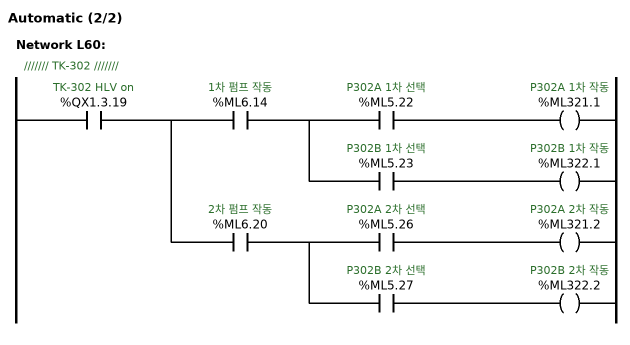
(* [picture p24: Automatic rungs L60-L60] *)
(* /////// TK-302 /////// *)
(* Rung L60 *)
%ML321.1 := %QX1.3.19 AND %ML6.14 AND %ML5.22;
%ML322.1 := %QX1.3.19 AND %ML6.14 AND %ML5.23;
%ML321.2 := %QX1.3.19 AND %ML6.20 AND %ML5.26;
%ML322.2 := %QX1.3.19 AND %ML6.20 AND %ML5.27;
END_PROGRAM

PROGRAM Analog (* task: 스캔 프로그램 *)
VAR_EXTERNAL
    _0100_CH0_ACT : BOOL; (* AT %UX1.0.16 *) (* 아날로그입력 모듈: 채널0 운전중 *)
    _0100_CH0_DATA : INT; (* AT %UW1.0.2 *) (* 아날로그입력 모듈: 채널0 변환값 *)
    _0100_CH0_IDD : BOOL; (* AT %UX1.0.160 *) (* 아날로그입력 모듈: 채널0 입력단선검출 *)
    _0100_CH1_ACT : BOOL; (* AT %UX1.0.17 *) (* 아날로그입력 모듈: 채널1 운전중 *)
    _0100_CH1_DATA : INT; (* AT %UW1.0.3 *) (* 아날로그입력 모듈: 채널1 변환값 *)
    _0100_CH1_IDD : BOOL; (* AT %UX1.0.161 *) (* 아날로그입력 모듈: 채널1 입력단선검출 *)
    _0100_CH2_ACT : BOOL; (* AT %UX1.0.18 *) (* 아날로그입력 모듈: 채널2 운전중 *)
    _0100_CH2_DATA : INT; (* AT %UW1.0.4 *) (* 아날로그입력 모듈: 채널2 변환값 *)
    _0100_CH2_IDD : BOOL; (* AT %UX1.0.162 *) (* 아날로그입력 모듈: 채널2 입력단선검출 *)
    _0100_CH3_ACT : BOOL; (* AT %UX1.0.19 *) (* 아날로그입력 모듈: 채널3 운전중 *)
    _0100_CH3_DATA : INT; (* AT %UW1.0.5 *) (* 아날로그입력 모듈: 채널3 변환값 *)
    _0100_CH3_IDD : BOOL; (* AT %UX1.0.163 *) (* 아날로그입력 모듈: 채널3 입력단선검출 *)
    _0100_CH4_ACT : BOOL; (* AT %UX1.0.20 *) (* 아날로그입력 모듈: 채널4 운전중 *)
    _0100_CH4_DATA : INT; (* AT %UW1.0.6 *) (* 아날로그입력 모듈: 채널4 변환값 *)
    _0100_CH4_IDD : BOOL; (* AT %UX1.0.164 *) (* 아날로그입력 모듈: 채널4 입력단선검출 *)
    _0100_CH5_ACT : BOOL; (* AT %UX1.0.21 *) (* 아날로그입력 모듈: 채널5 운전중 *)
    _0100_CH5_DATA : INT; (* AT %UW1.0.7 *) (* 아날로그입력 모듈: 채널5 변환값 *)
    _0100_CH5_IDD : BOOL; (* AT %UX1.0.165 *) (* 아날로그입력 모듈: 채널5 입력단선검출 *)
    _0100_CH6_ACT : BOOL; (* AT %UX1.0.22 *) (* 아날로그입력 모듈: 채널6 운전중 *)
    _0100_CH6_DATA : INT; (* AT %UW1.0.8 *) (* 아날로그입력 모듈: 채널6 변환값 *)
    _0100_CH6_IDD : BOOL; (* AT %UX1.0.166 *) (* 아날로그입력 모듈: 채널6 입력단선검출 *)
END_VAR
VAR
    _t1 : BOOL;
    _t2 : BOOL;
    _t3 : BOOL;
    _t4 : BOOL;
    _t5 : BOOL;
    _t6 : BOOL;
    _t7 : BOOL;
    _t8 : BOOL;
    _t9 : BOOL;
END_VAR

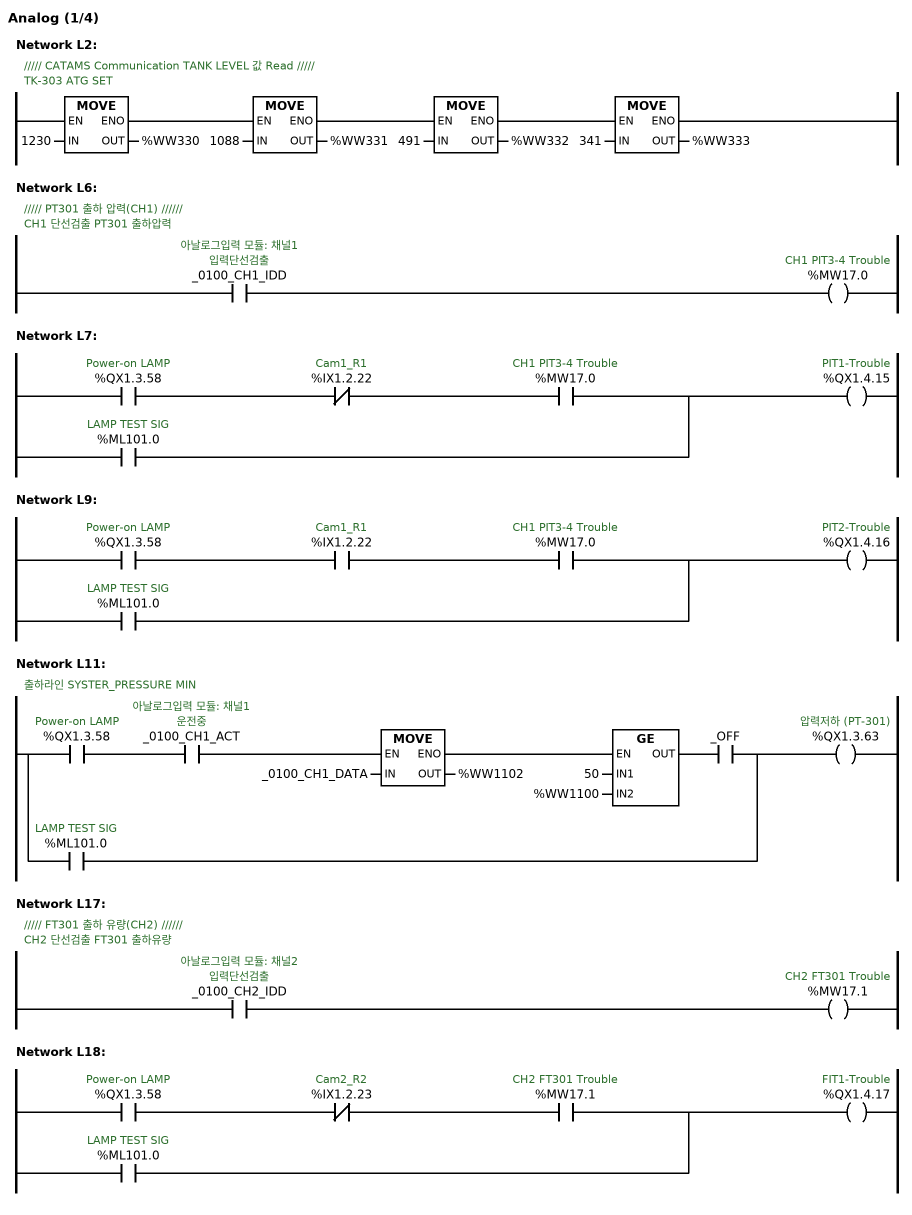
(* ///// CATAMS Communication TANK LEVEL 값 Read ///// *)
(* TK-303 ATG SET *)
(* Rung L2 *)
%WW330 := 1230;
%WW331 := 1088;
%WW332 := 491;
%WW333 := 341;
(* ///// PT301 출하 압력(CH1) ////// *)
(* Rung L6 *)
%MW17.0 := _0100_CH1_IDD;
(* CH1 단선검출 PT301 출하압력 *)
(* Rung L7 *)
%QX1.4.15 := (%QX1.3.58 AND NOT %IX1.2.22 AND %MW17.0) OR %ML101.0;
(* Rung L9 *)
%QX1.4.16 := (%QX1.3.58 AND %IX1.2.22 AND %MW17.0) OR %ML101.0;
(* Rung L11 *)
IF %QX1.3.58 AND _0100_CH1_ACT THEN
    %WW1102 := _0100_CH1_DATA;
    _t1 := 50 >= %WW1100;
END_IF;
%QX1.3.63 := (_t1 AND _OFF) OR %ML101.0;
(* 출하라인 SYSTER_PRESSURE MIN *)
(* ///// FT301 출하 유량(CH2) ////// *)
(* Rung L17 *)
%MW17.1 := _0100_CH2_IDD;
(* CH2 단선검출 FT301 출하유량 *)
(* Rung L18 *)
%QX1.4.17 := (%QX1.3.58 AND NOT %IX1.2.23 AND %MW17.1) OR %ML101.0;

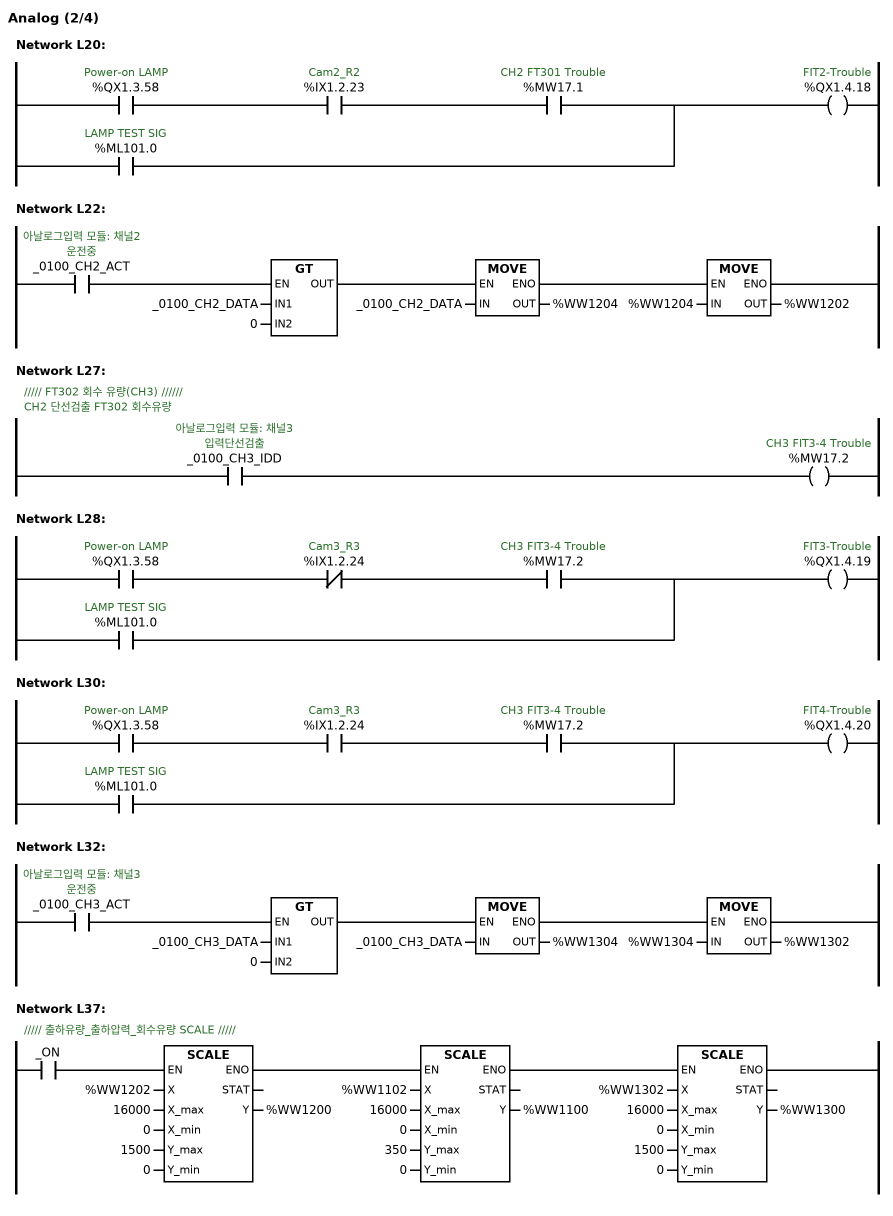
(* Rung L20 *)
%QX1.4.18 := (%QX1.3.58 AND %IX1.2.23 AND %MW17.1) OR %ML101.0;
(* Rung L22 *)
IF _0100_CH2_ACT THEN _t2 := _0100_CH2_DATA > 0; END_IF;
IF _t2 THEN
    %WW1204 := _0100_CH2_DATA;
    %WW1202 := %WW1204;
END_IF;
(* ///// FT302 회수 유량(CH3) ////// *)
(* Rung L27 *)
%MW17.2 := _0100_CH3_IDD;
(* CH2 단선검출 FT302 회수유량 *)
(* Rung L28 *)
%QX1.4.19 := (%QX1.3.58 AND NOT %IX1.2.24 AND %MW17.2) OR %ML101.0;
(* Rung L30 *)
%QX1.4.20 := (%QX1.3.58 AND %IX1.2.24 AND %MW17.2) OR %ML101.0;
(* Rung L32 *)
IF _0100_CH3_ACT THEN _t3 := _0100_CH3_DATA > 0; END_IF;
IF _t3 THEN
    %WW1304 := _0100_CH3_DATA;
    %WW1302 := %WW1304;
END_IF;
(* ///// 출하유량_출하압력_회수유량 SCALE ///// *)
(* Rung L37 *)
IF _ON THEN
    SCALE(X := %WW1202, X_max := 16000, X_min := 0, Y_max := 1500, Y_min := 0, Y => %WW1200);
    SCALE(X := %WW1102, X_max := 16000, X_min := 0, Y_max := 350, Y_min := 0, Y => %WW1100);
    SCALE(X := %WW1302, X_max := 16000, X_min := 0, Y_max := 1500, Y_min := 0, Y => %WW1300);
END_IF;

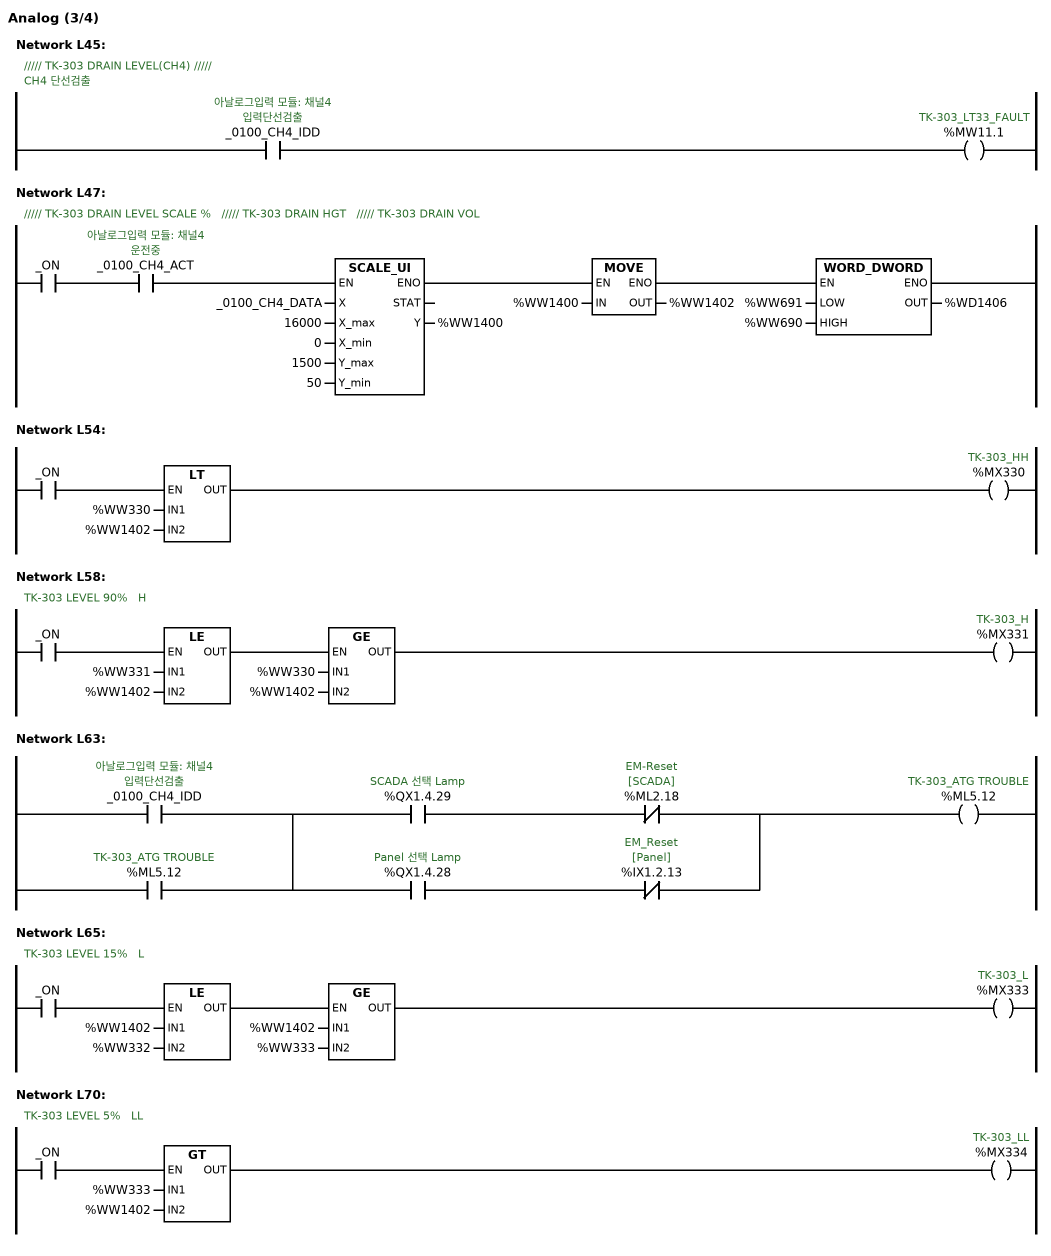
(* ///// TK-303 DRAIN LEVEL(CH4) ///// *)
(* Rung L45 *)
%MW11.1 := _0100_CH4_IDD;
(* CH4 단선검출 *)
(* ///// TK-303 DRAIN LEVEL SCALE %   ///// TK-303 DRAIN HGT   ///// TK-303 DRAIN VOL *)
(* Rung L47 *)
IF _ON AND _0100_CH4_ACT THEN
    SCALE_UI(X := _0100_CH4_DATA, X_max := 16000, X_min := 0, Y_max := 1500, Y_min := 50, Y => %WW1400);
    %WW1402 := %WW1400;
    %WD1406 := WORD_DWORD(LOW := %WW691, HIGH := %WW690);
END_IF;
(* Rung L54 *)
IF _ON THEN _t4 := %WW330 < %WW1402; END_IF;
%MX330 := _t4;
(* Rung L58 *)
IF _ON THEN _t5 := %WW331 <= %WW1402; END_IF;
IF _t5 THEN _t6 := %WW330 >= %WW1402; END_IF;
%MX331 := _t6;
(* TK-303 LEVEL 90%   H *)
(* Rung L63 *)
%ML5.12 := (_0100_CH4_IDD OR %ML5.12) AND ((%QX1.4.29 AND NOT %ML2.18) OR (%QX1.4.28 AND NOT %IX1.2.13));
(* Rung L65 *)
IF _ON THEN _t7 := %WW1402 <= %WW332; END_IF;
IF _t7 THEN _t8 := %WW1402 >= %WW333; END_IF;
%MX333 := _t8;
(* TK-303 LEVEL 15%   L *)
(* Rung L70 *)
IF _ON THEN _t9 := %WW333 > %WW1402; END_IF;
%MX334 := _t9;
(* TK-303 LEVEL 5%   LL *)

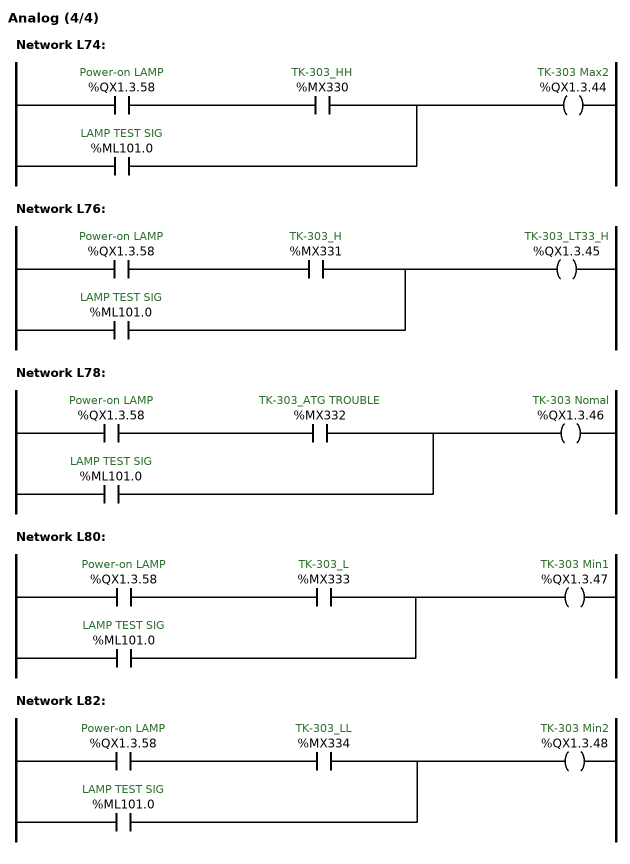
(* Rung L74 *)
%QX1.3.44 := (%QX1.3.58 AND %MX330) OR %ML101.0;
(* Rung L76 *)
%QX1.3.45 := (%QX1.3.58 AND %MX331) OR %ML101.0;
(* Rung L78 *)
%QX1.3.46 := (%QX1.3.58 AND %MX332) OR %ML101.0;
(* Rung L80 *)
%QX1.3.47 := (%QX1.3.58 AND %MX333) OR %ML101.0;
(* Rung L82 *)
%QX1.3.48 := (%QX1.3.58 AND %MX334) OR %ML101.0;
END_PROGRAM

PROGRAM Communiction (* task: 스캔 프로그램 *)
VAR
    C0010 : CTR; (* 통신 *)
    C19_TLV_OFD : TOF;
    C20_TLV_OFD : TOF;
    C21_TLV_OFD : TOF;
    C22_TLV_OFD : TOF;
    C23_TLV_OFD : TOF;
    C24_TLV_OFD : TOF;
    C24_TLV_OFD1 : TON;
    C24_TLV_OFD2 : TON;
    C24_TLV_OFD3 : TOF;
    C24_TLV_OFD4 : TOF;
    C24_TLV_OFD5 : TON;
    CTR10 : BOOL; (* 모드버스 송신블럭 번호 *)
END_VAR
VAR_EXTERNAL
    _0100_CH1_ACT : BOOL; (* AT %UX1.0.17 *) (* 아날로그입력 모듈: 채널1 운전중 *)
    _0100_CH1_DATA : INT; (* AT %UW1.0.3 *) (* 아날로그입력 모듈: 채널1 변환값 *)
END_VAR
VAR
    _t1 : BOOL;
    _t2 : BOOL;
    _t3 : BOOL;
    _t4 : BOOL;
    _t5 : BOOL;
    _t6 : BOOL;
    _t7 : BOOL;
    _t8 : BOOL;
    _t9 : BOOL;
    _t10 : BOOL;
    _t11 : BOOL;
    _t12 : BOOL;
    _t13 : BOOL;
    _t14 : BOOL;
END_VAR

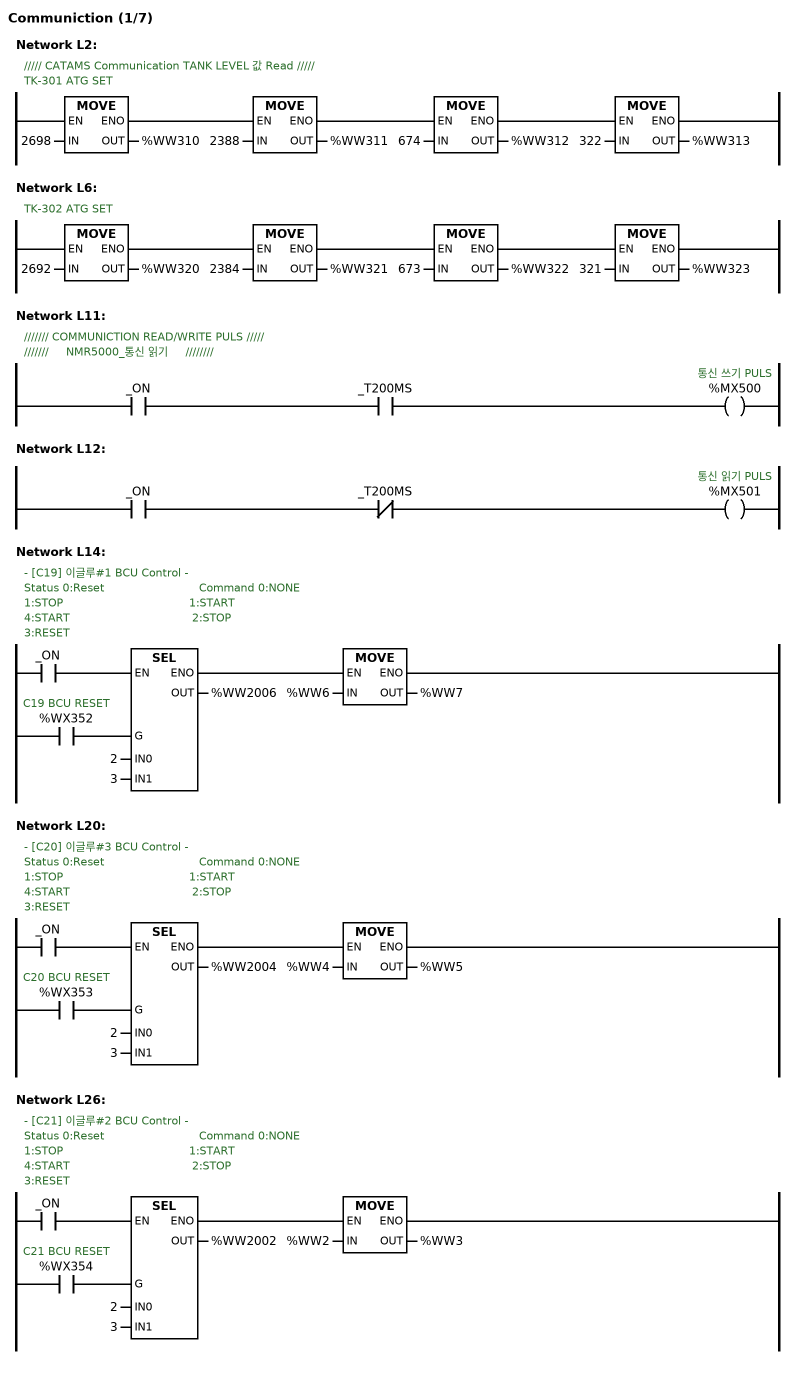
(* ///// CATAMS Communication TANK LEVEL 값 Read ///// *)
(* TK-301 ATG SET *)
(* Rung L2 *)
%WW310 := 2698;
%WW311 := 2388;
%WW312 := 674;
%WW313 := 322;
(* TK-302 ATG SET *)
(* Rung L6 *)
%WW320 := 2692;
%WW321 := 2384;
%WW322 := 673;
%WW323 := 321;
(* /////// COMMUNICTION READ/WRITE PULS ///// *)
(* ///////     NMR5000_통신 읽기     //////// *)
(* Rung L11 *)
%MX500 := _ON AND _T200MS;
(* Rung L12 *)
%MX501 := _ON AND NOT _T200MS;
(* - [C19] 이글루#1 BCU Control - / Status 0:Reset                           Command 0:NONE / 1:STOP                                    1:START / 4:START                                   2:STOP / 3:RESET *)
(* Rung L14 *)
IF _ON THEN
    %WW2006 := SEL(G := %WX352, IN0 := 2, IN1 := 3);
    %WW7 := %WW6;
END_IF;
(* - [C20] 이글루#3 BCU Control - / Status 0:Reset                           Command 0:NONE / 1:STOP                                    1:START / 4:START                                   2:STOP / 3:RESET *)
(* Rung L20 *)
IF _ON THEN
    %WW2004 := SEL(G := %WX353, IN0 := 2, IN1 := 3);
    %WW5 := %WW4;
END_IF;
(* - [C21] 이글루#2 BCU Control - / Status 0:Reset                           Command 0:NONE / 1:STOP                                    1:START / 4:START                                   2:STOP / 3:RESET *)
(* Rung L26 *)
IF _ON THEN
    %WW2002 := SEL(G := %WX354, IN0 := 2, IN1 := 3);
    %WW3 := %WW2;
END_IF;

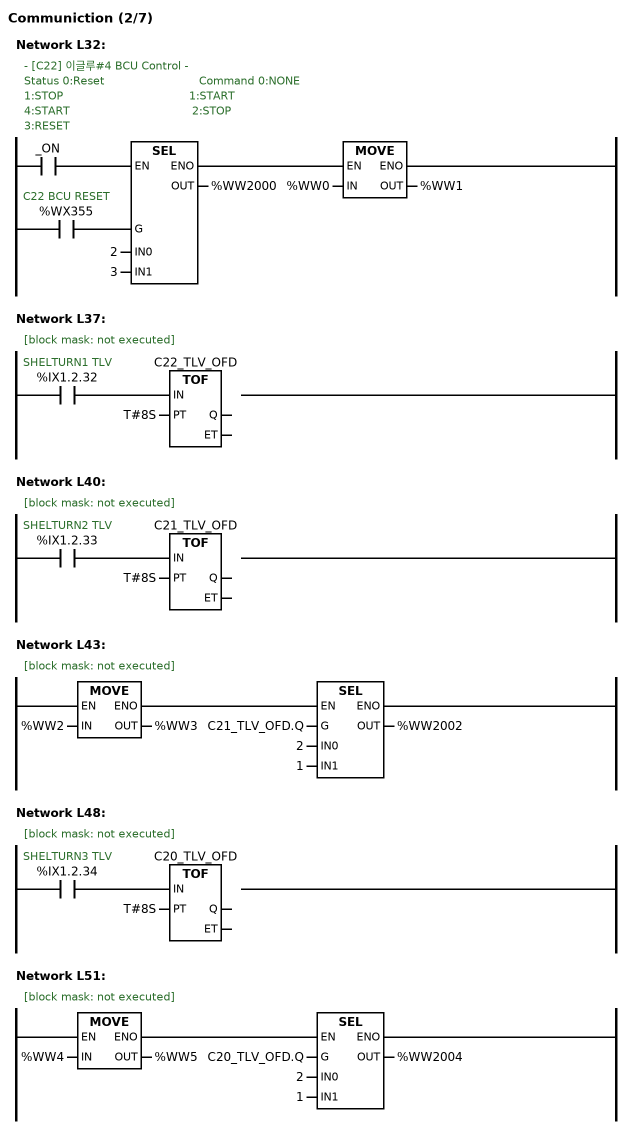
(* - [C22] 이글루#4 BCU Control - / Status 0:Reset                           Command 0:NONE / 1:STOP                                    1:START / 4:START                                   2:STOP / 3:RESET *)
(* Rung L32 *)
IF _ON THEN
    %WW2000 := SEL(G := %WX355, IN0 := 2, IN1 := 3);
    %WW1 := %WW0;
END_IF;
(* Rung L37 is block-masked: not executed *)
// C22_TLV_OFD(IN := %IX1.2.32, PT := T#8S);
(* Rung L40 is block-masked: not executed *)
// C21_TLV_OFD(IN := %IX1.2.33, PT := T#8S);
(* Rung L43 is block-masked: not executed *)
// %WW3 := %WW2;
// %WW2002 := SEL(G := C21_TLV_OFD.Q, IN0 := 2, IN1 := 1);
(* Rung L48 is block-masked: not executed *)
// C20_TLV_OFD(IN := %IX1.2.34, PT := T#8S);
(* Rung L51 is block-masked: not executed *)
// %WW5 := %WW4;
// %WW2004 := SEL(G := C20_TLV_OFD.Q, IN0 := 2, IN1 := 1);

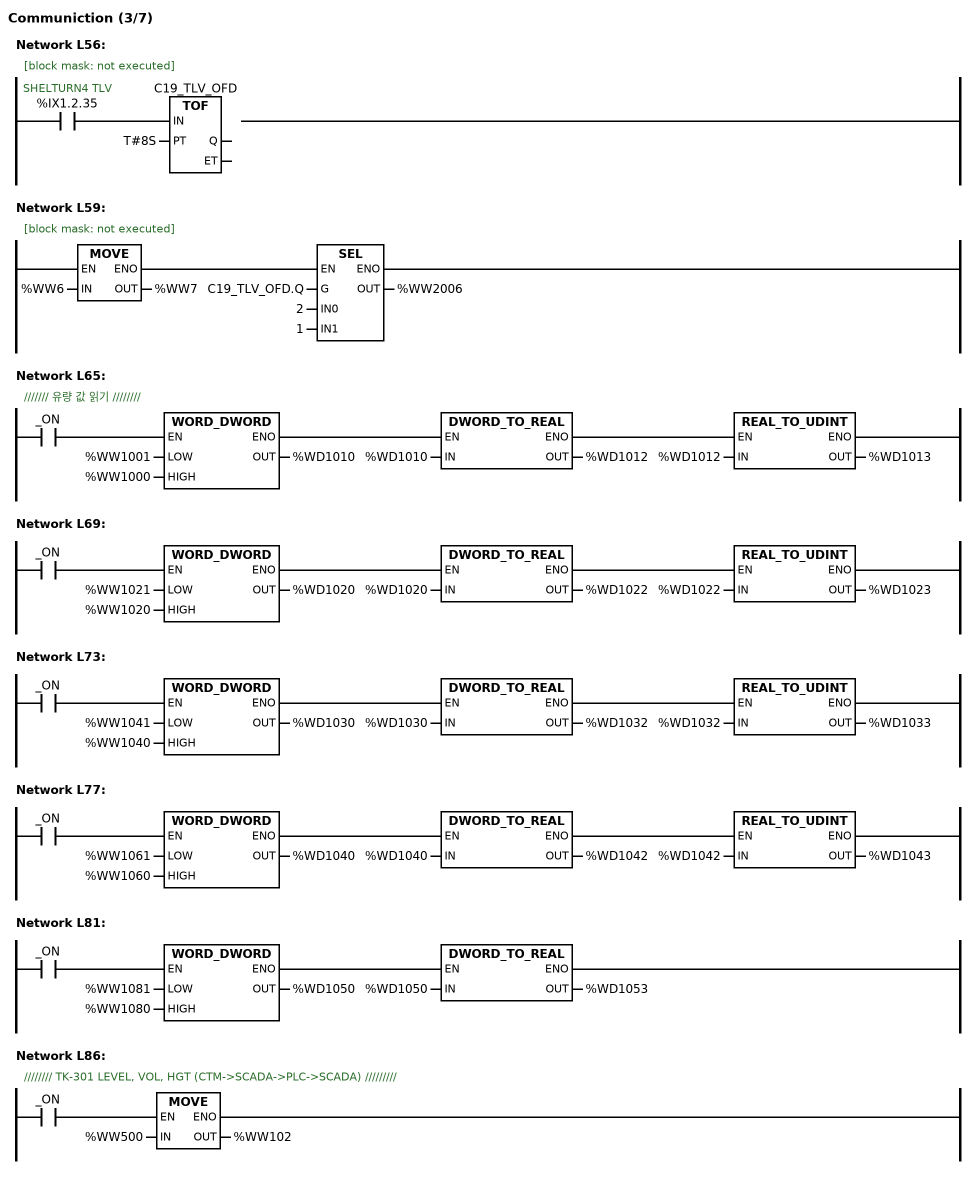
(* Rung L56 is block-masked: not executed *)
// C19_TLV_OFD(IN := %IX1.2.35, PT := T#8S);
(* Rung L59 is block-masked: not executed *)
// %WW7 := %WW6;
// %WW2006 := SEL(G := C19_TLV_OFD.Q, IN0 := 2, IN1 := 1);
(* /////// 유량 값 읽기 //////// *)
(* Rung L65 *)
IF _ON THEN
    %WD1010 := WORD_DWORD(LOW := %WW1001, HIGH := %WW1000);
    %WD1012 := DWORD_TO_REAL(%WD1010);
    %WD1013 := REAL_TO_UDINT(%WD1012);
END_IF;
(* Rung L69 *)
IF _ON THEN
    %WD1020 := WORD_DWORD(LOW := %WW1021, HIGH := %WW1020);
    %WD1022 := DWORD_TO_REAL(%WD1020);
    %WD1023 := REAL_TO_UDINT(%WD1022);
END_IF;
(* Rung L73 *)
IF _ON THEN
    %WD1030 := WORD_DWORD(LOW := %WW1041, HIGH := %WW1040);
    %WD1032 := DWORD_TO_REAL(%WD1030);
    %WD1033 := REAL_TO_UDINT(%WD1032);
END_IF;
(* Rung L77 *)
IF _ON THEN
    %WD1040 := WORD_DWORD(LOW := %WW1061, HIGH := %WW1060);
    %WD1042 := DWORD_TO_REAL(%WD1040);
    %WD1043 := REAL_TO_UDINT(%WD1042);
END_IF;
(* Rung L81 *)
IF _ON THEN
    %WD1050 := WORD_DWORD(LOW := %WW1081, HIGH := %WW1080);
    %WD1053 := DWORD_TO_REAL(%WD1050);
END_IF;
(* //////// TK-301 LEVEL, VOL, HGT (CTM->SCADA->PLC->SCADA) ///////// *)
(* Rung L86 *)
IF _ON THEN %WW102 := %WW500; END_IF;

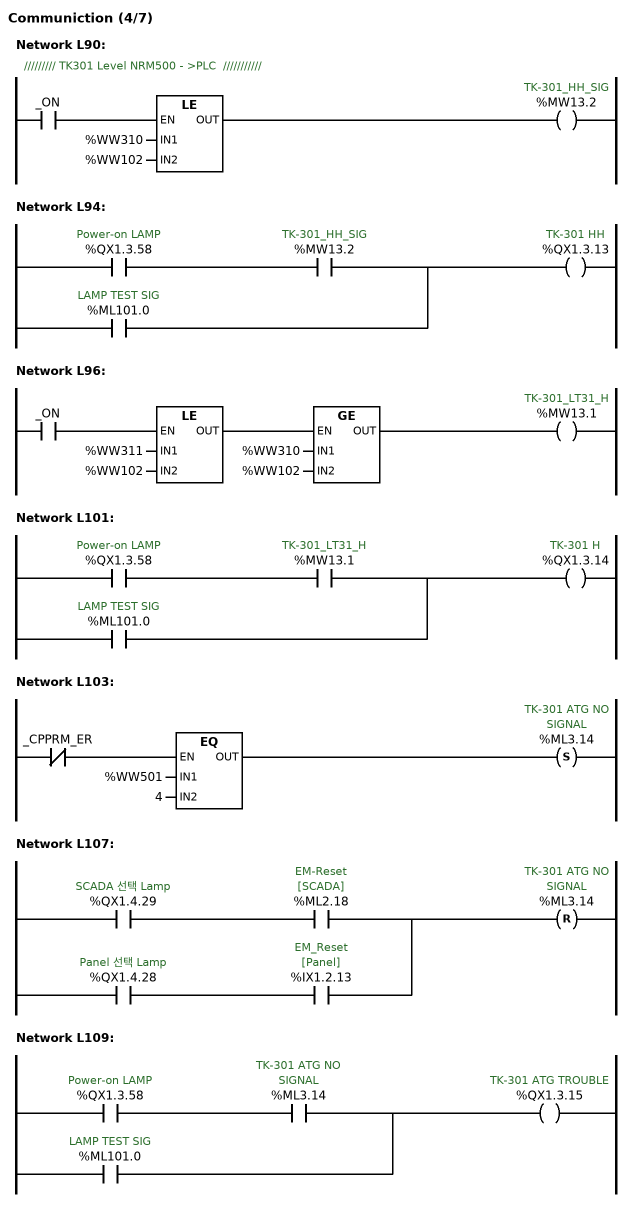
(* ///////// TK301 Level NRM500 - >PLC  /////////// *)
(* Rung L90 *)
IF _ON THEN _t1 := %WW310 <= %WW102; END_IF;
%MW13.2 := _t1;
(* Rung L94 *)
%QX1.3.13 := (%QX1.3.58 AND %MW13.2) OR %ML101.0;
(* Rung L96 *)
IF _ON THEN _t2 := %WW311 <= %WW102; END_IF;
IF _t2 THEN _t3 := %WW310 >= %WW102; END_IF;
%MW13.1 := _t3;
(* Rung L101 *)
%QX1.3.14 := (%QX1.3.58 AND %MW13.1) OR %ML101.0;
(* Rung L103 *)
IF NOT _CPPRM_ER THEN _t4 := %WW501 = 4; END_IF;
IF _t4 THEN %ML3.14 := TRUE; END_IF;
(* Rung L107 *)
IF (%QX1.4.29 AND %ML2.18) OR (%QX1.4.28 AND %IX1.2.13) THEN %ML3.14 := FALSE; END_IF;
(* Rung L109 *)
%QX1.3.15 := (%QX1.3.58 AND %ML3.14) OR %ML101.0;

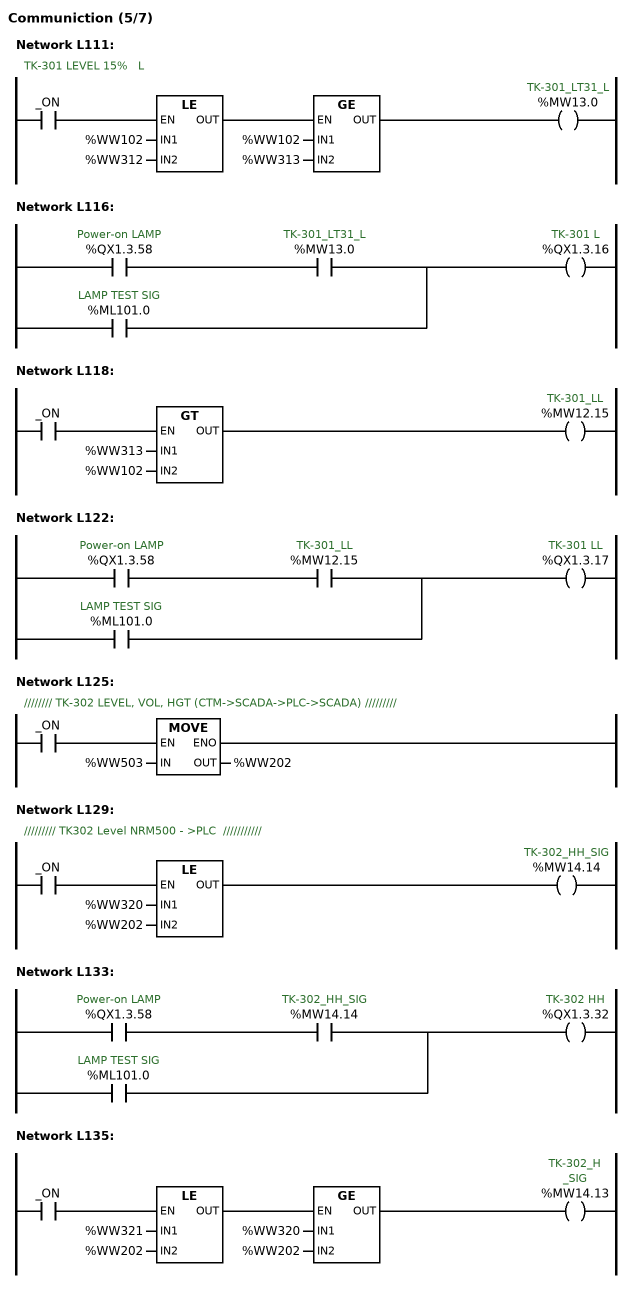
(* Rung L111 *)
IF _ON THEN _t5 := %WW102 <= %WW312; END_IF;
IF _t5 THEN _t6 := %WW102 >= %WW313; END_IF;
%MW13.0 := _t6;
(* TK-301 LEVEL 15%   L *)
(* Rung L116 *)
%QX1.3.16 := (%QX1.3.58 AND %MW13.0) OR %ML101.0;
(* Rung L118 *)
IF _ON THEN _t7 := %WW313 > %WW102; END_IF;
%MW12.15 := _t7;
(* Rung L122 *)
%QX1.3.17 := (%QX1.3.58 AND %MW12.15) OR %ML101.0;
(* //////// TK-302 LEVEL, VOL, HGT (CTM->SCADA->PLC->SCADA) ///////// *)
(* Rung L125 *)
IF _ON THEN %WW202 := %WW503; END_IF;
(* ///////// TK302 Level NRM500 - >PLC  /////////// *)
(* Rung L129 *)
IF _ON THEN _t8 := %WW320 <= %WW202; END_IF;
%MW14.14 := _t8;
(* Rung L133 *)
%QX1.3.32 := (%QX1.3.58 AND %MW14.14) OR %ML101.0;
(* Rung L135 *)
IF _ON THEN _t9 := %WW321 <= %WW202; END_IF;
IF _t9 THEN _t10 := %WW320 >= %WW202; END_IF;
%MW14.13 := _t10;

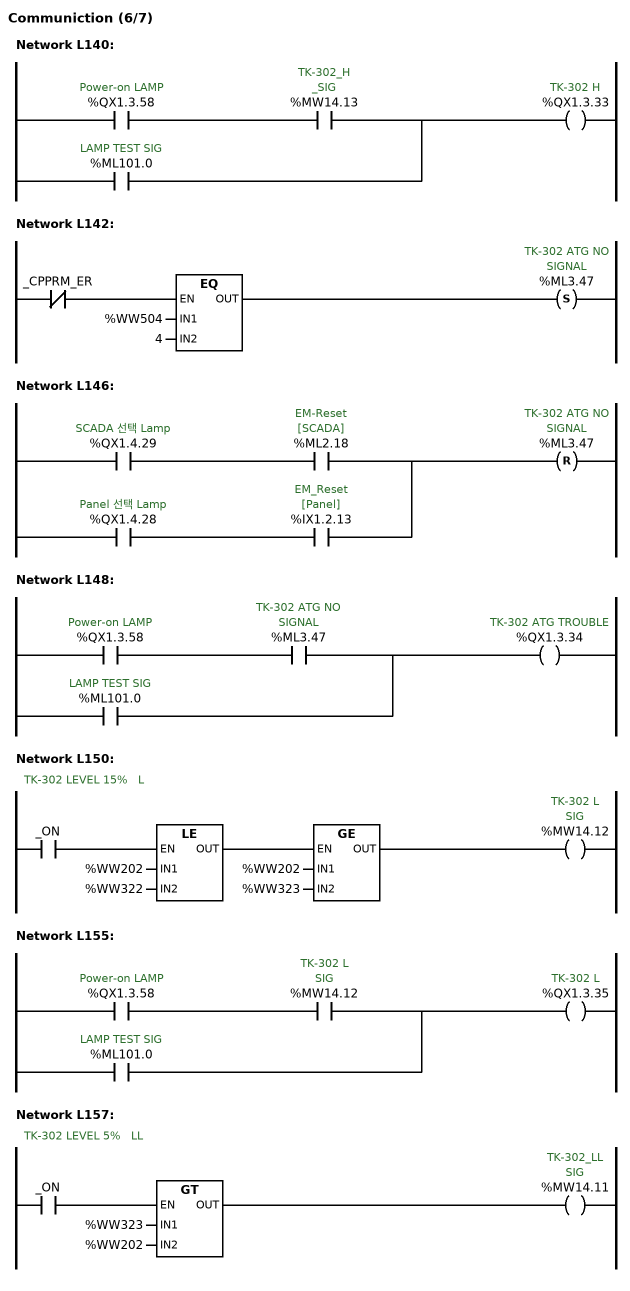
(* Rung L140 *)
%QX1.3.33 := (%QX1.3.58 AND %MW14.13) OR %ML101.0;
(* Rung L142 *)
IF NOT _CPPRM_ER THEN _t11 := %WW504 = 4; END_IF;
IF _t11 THEN %ML3.47 := TRUE; END_IF;
(* Rung L146 *)
IF (%QX1.4.29 AND %ML2.18) OR (%QX1.4.28 AND %IX1.2.13) THEN %ML3.47 := FALSE; END_IF;
(* Rung L148 *)
%QX1.3.34 := (%QX1.3.58 AND %ML3.47) OR %ML101.0;
(* Rung L150 *)
IF _ON THEN _t12 := %WW202 <= %WW322; END_IF;
IF _t12 THEN _t13 := %WW202 >= %WW323; END_IF;
%MW14.12 := _t13;
(* TK-302 LEVEL 15%   L *)
(* Rung L155 *)
%QX1.3.35 := (%QX1.3.58 AND %MW14.12) OR %ML101.0;
(* Rung L157 *)
IF _ON THEN _t14 := %WW323 > %WW202; END_IF;
%MW14.11 := _t14;
(* TK-302 LEVEL 5%   LL *)

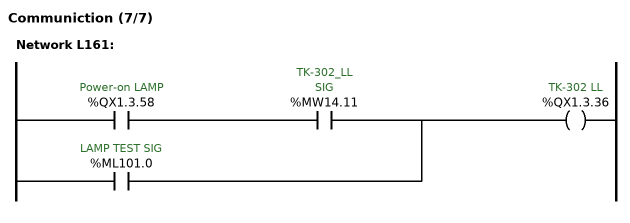
(* Rung L161 *)
%QX1.3.36 := (%QX1.3.58 AND %MW14.11) OR %ML101.0;
END_PROGRAM

PROGRAM Scada (* task: 스캔 프로그램 *)
VAR
    T1 : BOOL;
    T9 : TON;
END_VAR

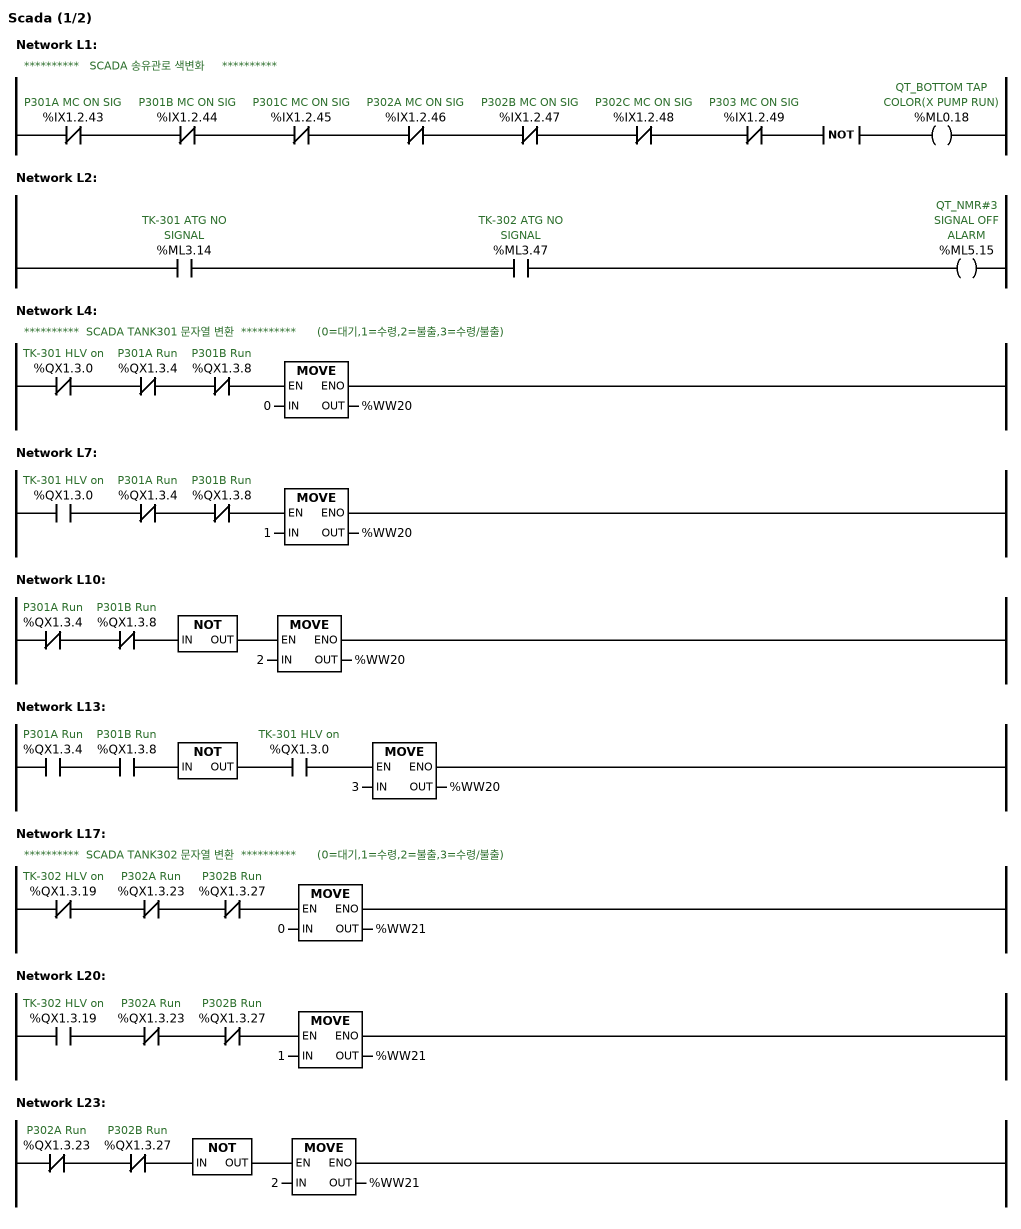
(* **********   SCADA 송유관로 색변화     ********** *)
(* Rung L1 *)
%ML0.18 := NOT (NOT %IX1.2.43 AND NOT %IX1.2.44 AND NOT %IX1.2.45 AND NOT %IX1.2.46 AND NOT %IX1.2.47 AND NOT %IX1.2.48 AND NOT %IX1.2.49);
(* Rung L2 *)
%ML5.15 := %ML3.14 AND %ML3.47;
(* **********  SCADA TANK301 문자열 변환  **********      (0=대기,1=수령,2=불출,3=수령/불출) *)
(* Rung L4 *)
IF NOT %QX1.3.0 AND NOT %QX1.3.4 AND NOT %QX1.3.8 THEN %WW20 := 0; END_IF;
(* Rung L7 *)
IF %QX1.3.0 AND NOT %QX1.3.4 AND NOT %QX1.3.8 THEN %WW20 := 1; END_IF;
(* Rung L10 *)
IF NOT (NOT %QX1.3.4 AND NOT %QX1.3.8) THEN %WW20 := 2; END_IF;
(* Rung L13 *)
IF (NOT (%QX1.3.4 AND %QX1.3.8)) AND %QX1.3.0 THEN %WW20 := 3; END_IF;
(* **********  SCADA TANK302 문자열 변환  **********      (0=대기,1=수령,2=불출,3=수령/불출) *)
(* Rung L17 *)
IF NOT %QX1.3.19 AND NOT %QX1.3.23 AND NOT %QX1.3.27 THEN %WW21 := 0; END_IF;
(* Rung L20 *)
IF %QX1.3.19 AND NOT %QX1.3.23 AND NOT %QX1.3.27 THEN %WW21 := 1; END_IF;
(* Rung L23 *)
IF NOT (NOT %QX1.3.23 AND NOT %QX1.3.27) THEN %WW21 := 2; END_IF;

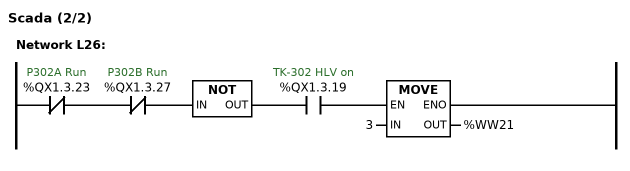
(* Rung L26 *)
IF (NOT (NOT %QX1.3.23 AND NOT %QX1.3.27)) AND %QX1.3.19 THEN %WW21 := 3; END_IF;
END_PROGRAM

PROGRAM Setting (* task: 스캔 프로그램 *)
VAR
    _t1 : BOOL;
    _t2 : BOOL;
    _t3 : BOOL;
    _t4 : BOOL;
    _t5 : BOOL;
    _t6 : BOOL;
    _t7 : BOOL;
    _t8 : BOOL;
END_VAR

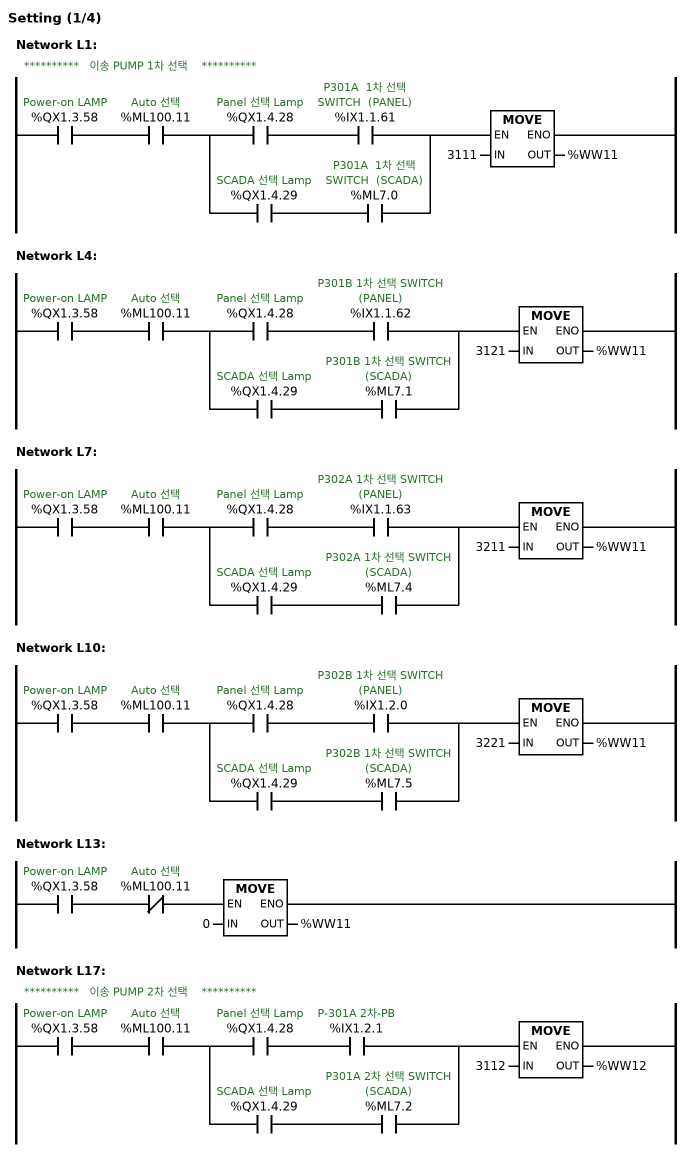
(* **********   이송 PUMP 1차 선택    ********** *)
(* Rung L1 *)
IF %QX1.3.58 AND %ML100.11 AND ((%QX1.4.28 AND %IX1.1.61) OR (%QX1.4.29 AND %ML7.0)) THEN
    %WW11 := 3111;
END_IF;
(* Rung L4 *)
IF %QX1.3.58 AND %ML100.11 AND ((%QX1.4.28 AND %IX1.1.62) OR (%QX1.4.29 AND %ML7.1)) THEN
    %WW11 := 3121;
END_IF;
(* Rung L7 *)
IF %QX1.3.58 AND %ML100.11 AND ((%QX1.4.28 AND %IX1.1.63) OR (%QX1.4.29 AND %ML7.4)) THEN
    %WW11 := 3211;
END_IF;
(* Rung L10 *)
IF %QX1.3.58 AND %ML100.11 AND ((%QX1.4.28 AND %IX1.2.0) OR (%QX1.4.29 AND %ML7.5)) THEN
    %WW11 := 3221;
END_IF;
(* Rung L13 *)
IF %QX1.3.58 AND NOT %ML100.11 THEN %WW11 := 0; END_IF;
(* **********   이송 PUMP 2차 선택    ********** *)
(* Rung L17 *)
IF %QX1.3.58 AND %ML100.11 AND ((%QX1.4.28 AND %IX1.2.1) OR (%QX1.4.29 AND %ML7.2)) THEN
    %WW12 := 3112;
END_IF;

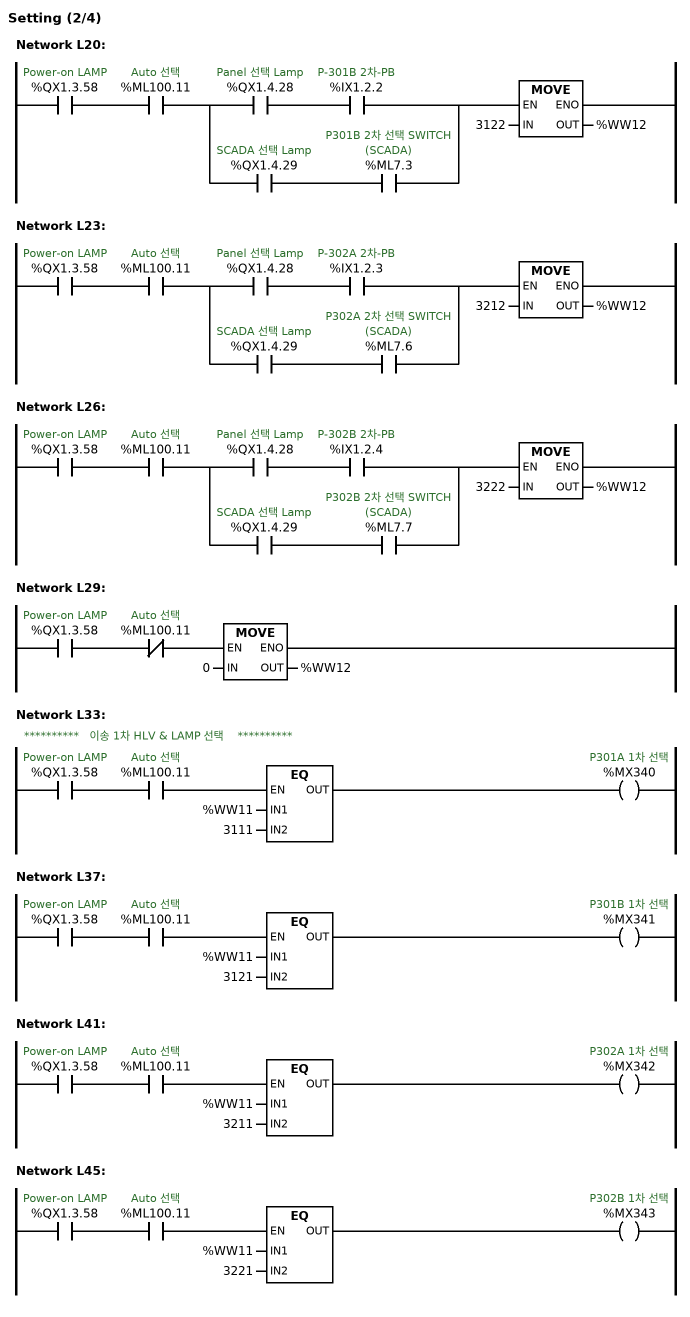
(* Rung L20 *)
IF %QX1.3.58 AND %ML100.11 AND ((%QX1.4.28 AND %IX1.2.2) OR (%QX1.4.29 AND %ML7.3)) THEN
    %WW12 := 3122;
END_IF;
(* Rung L23 *)
IF %QX1.3.58 AND %ML100.11 AND ((%QX1.4.28 AND %IX1.2.3) OR (%QX1.4.29 AND %ML7.6)) THEN
    %WW12 := 3212;
END_IF;
(* Rung L26 *)
IF %QX1.3.58 AND %ML100.11 AND ((%QX1.4.28 AND %IX1.2.4) OR (%QX1.4.29 AND %ML7.7)) THEN
    %WW12 := 3222;
END_IF;
(* Rung L29 *)
IF %QX1.3.58 AND NOT %ML100.11 THEN %WW12 := 0; END_IF;
(* **********   이송 1차 HLV & LAMP 선택    ********** *)
(* Rung L33 *)
IF %QX1.3.58 AND %ML100.11 THEN _t1 := %WW11 = 3111; END_IF;
%MX340 := _t1;
(* Rung L37 *)
IF %QX1.3.58 AND %ML100.11 THEN _t2 := %WW11 = 3121; END_IF;
%MX341 := _t2;
(* Rung L41 *)
IF %QX1.3.58 AND %ML100.11 THEN _t3 := %WW11 = 3211; END_IF;
%MX342 := _t3;
(* Rung L45 *)
IF %QX1.3.58 AND %ML100.11 THEN _t4 := %WW11 = 3221; END_IF;
%MX343 := _t4;

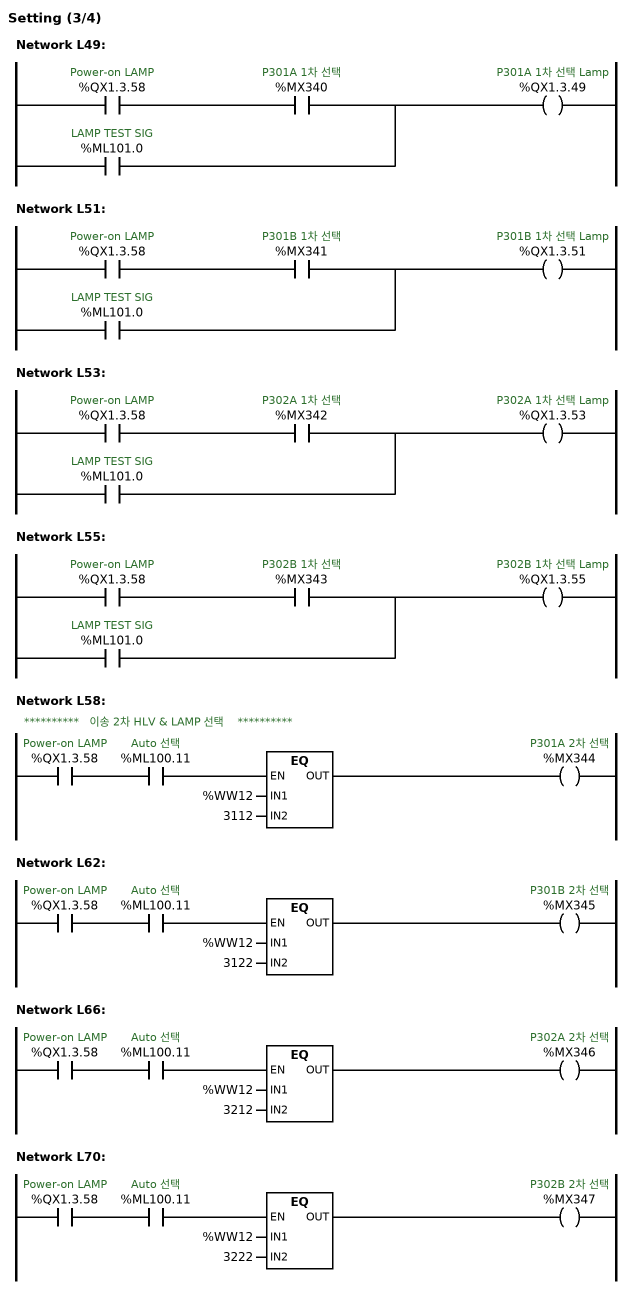
(* Rung L49 *)
%QX1.3.49 := (%QX1.3.58 AND %MX340) OR %ML101.0;
(* Rung L51 *)
%QX1.3.51 := (%QX1.3.58 AND %MX341) OR %ML101.0;
(* Rung L53 *)
%QX1.3.53 := (%QX1.3.58 AND %MX342) OR %ML101.0;
(* Rung L55 *)
%QX1.3.55 := (%QX1.3.58 AND %MX343) OR %ML101.0;
(* **********   이송 2차 HLV & LAMP 선택    ********** *)
(* Rung L58 *)
IF %QX1.3.58 AND %ML100.11 THEN _t5 := %WW12 = 3112; END_IF;
%MX344 := _t5;
(* Rung L62 *)
IF %QX1.3.58 AND %ML100.11 THEN _t6 := %WW12 = 3122; END_IF;
%MX345 := _t6;
(* Rung L66 *)
IF %QX1.3.58 AND %ML100.11 THEN _t7 := %WW12 = 3212; END_IF;
%MX346 := _t7;
(* Rung L70 *)
IF %QX1.3.58 AND %ML100.11 THEN _t8 := %WW12 = 3222; END_IF;
%MX347 := _t8;

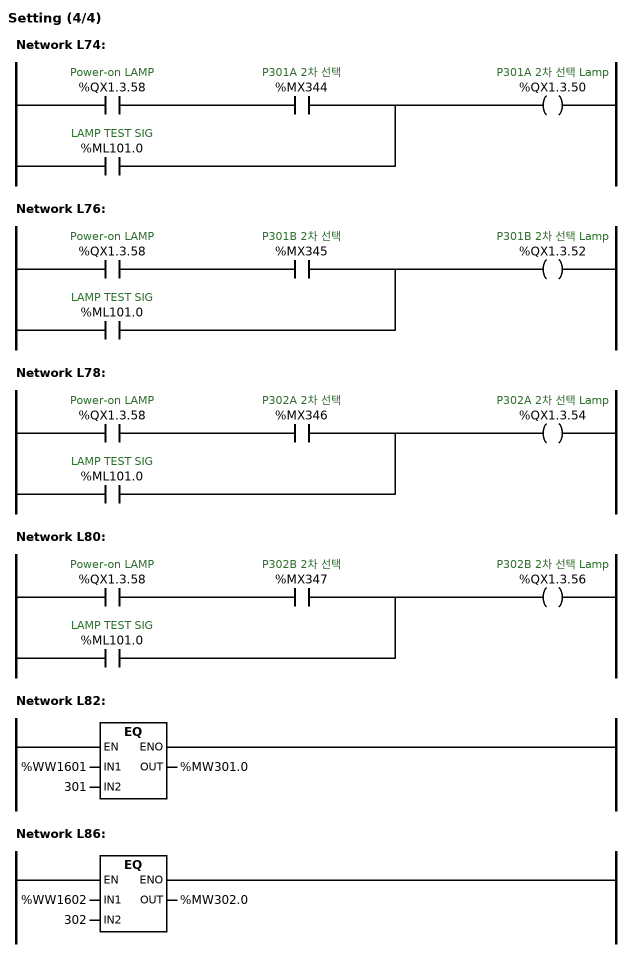
(* Rung L74 *)
%QX1.3.50 := (%QX1.3.58 AND %MX344) OR %ML101.0;
(* Rung L76 *)
%QX1.3.52 := (%QX1.3.58 AND %MX345) OR %ML101.0;
(* Rung L78 *)
%QX1.3.54 := (%QX1.3.58 AND %MX346) OR %ML101.0;
(* Rung L80 *)
%QX1.3.56 := (%QX1.3.58 AND %MX347) OR %ML101.0;
(* Rung L82 *)
%MW301.0 := %WW1601 = 301;
(* Rung L86 *)
%MW302.0 := %WW1602 = 302;
END_PROGRAM

PROGRAM Alarm (* task: 스캔 프로그램 *)
VAR_EXTERNAL
    C485 : TON;
    C486 : TON;
    C487 : TON;
    TCPIP : TON;
    _0000_STAND_ALONE : BOOL; (* AT %LX60144 *) (* FEnet: 연결 안된 상태(Ver 6.0이상) *)
END_VAR
VAR
    P301B_FS : TON;
    T20 : TON; (* Reset *)
    T8 : TON; (* Horn_off time *)
END_VAR

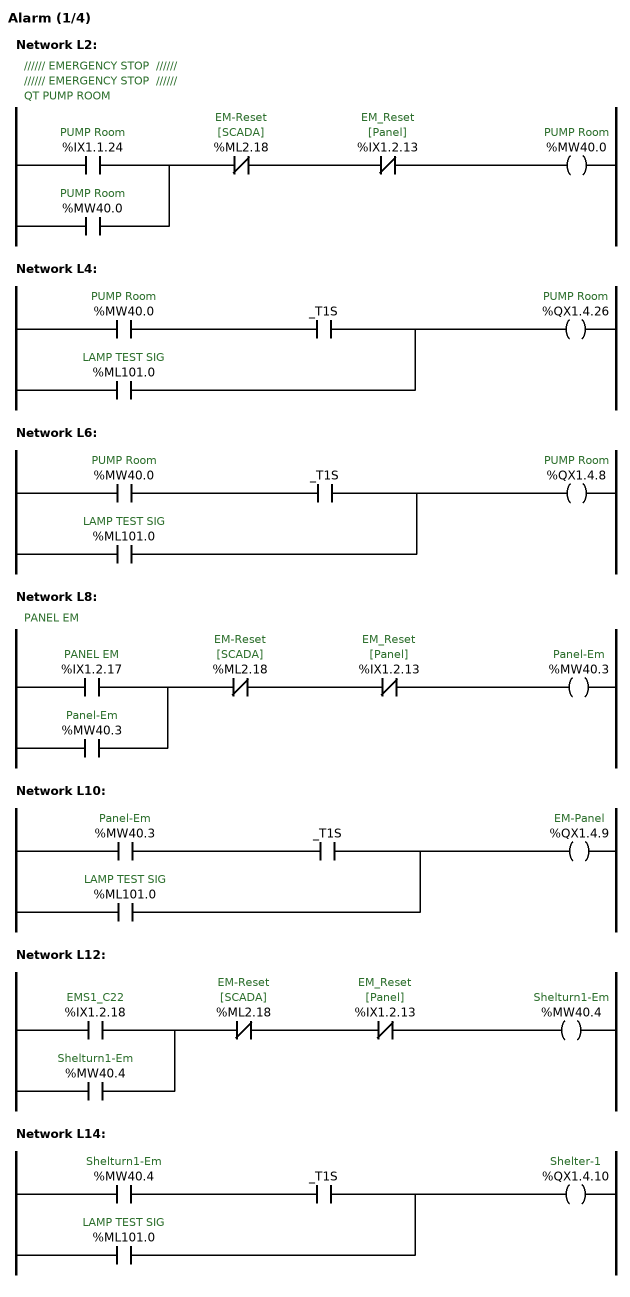
(* ////// EMERGENCY STOP  ////// *)
(* ////// EMERGENCY STOP  ////// *)
(* Rung L2 *)
%MW40.0 := (%IX1.1.24 OR %MW40.0) AND NOT %ML2.18 AND NOT %IX1.2.13;
(* QT PUMP ROOM *)
(* Rung L4 *)
%QX1.4.26 := (%MW40.0 AND _T1S) OR %ML101.0;
(* Rung L6 *)
%QX1.4.8 := (%MW40.0 AND _T1S) OR %ML101.0;
(* Rung L8 *)
%MW40.3 := (%IX1.2.17 OR %MW40.3) AND NOT %ML2.18 AND NOT %IX1.2.13;
(* PANEL EM *)
(* Rung L10 *)
%QX1.4.9 := (%MW40.3 AND _T1S) OR %ML101.0;
(* Rung L12 *)
%MW40.4 := (%IX1.2.18 OR %MW40.4) AND NOT %ML2.18 AND NOT %IX1.2.13;
(* Rung L14 *)
%QX1.4.10 := (%MW40.4 AND _T1S) OR %ML101.0;

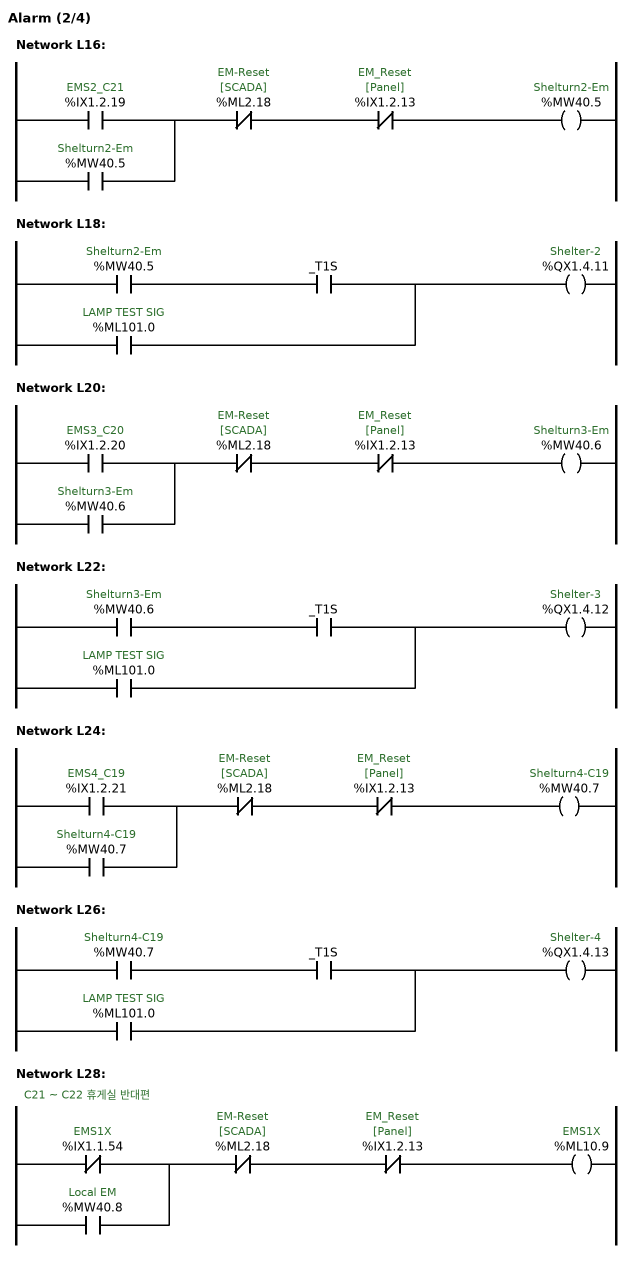
(* Rung L16 *)
%MW40.5 := (%IX1.2.19 OR %MW40.5) AND NOT %ML2.18 AND NOT %IX1.2.13;
(* Rung L18 *)
%QX1.4.11 := (%MW40.5 AND _T1S) OR %ML101.0;
(* Rung L20 *)
%MW40.6 := (%IX1.2.20 OR %MW40.6) AND NOT %ML2.18 AND NOT %IX1.2.13;
(* Rung L22 *)
%QX1.4.12 := (%MW40.6 AND _T1S) OR %ML101.0;
(* Rung L24 *)
%MW40.7 := (%IX1.2.21 OR %MW40.7) AND NOT %ML2.18 AND NOT %IX1.2.13;
(* Rung L26 *)
%QX1.4.13 := (%MW40.7 AND _T1S) OR %ML101.0;
(* Rung L28 *)
%ML10.9 := (NOT %IX1.1.54 OR %MW40.8) AND NOT %ML2.18 AND NOT %IX1.2.13;
(* C21 ~ C22 휴게실 반대편 *)

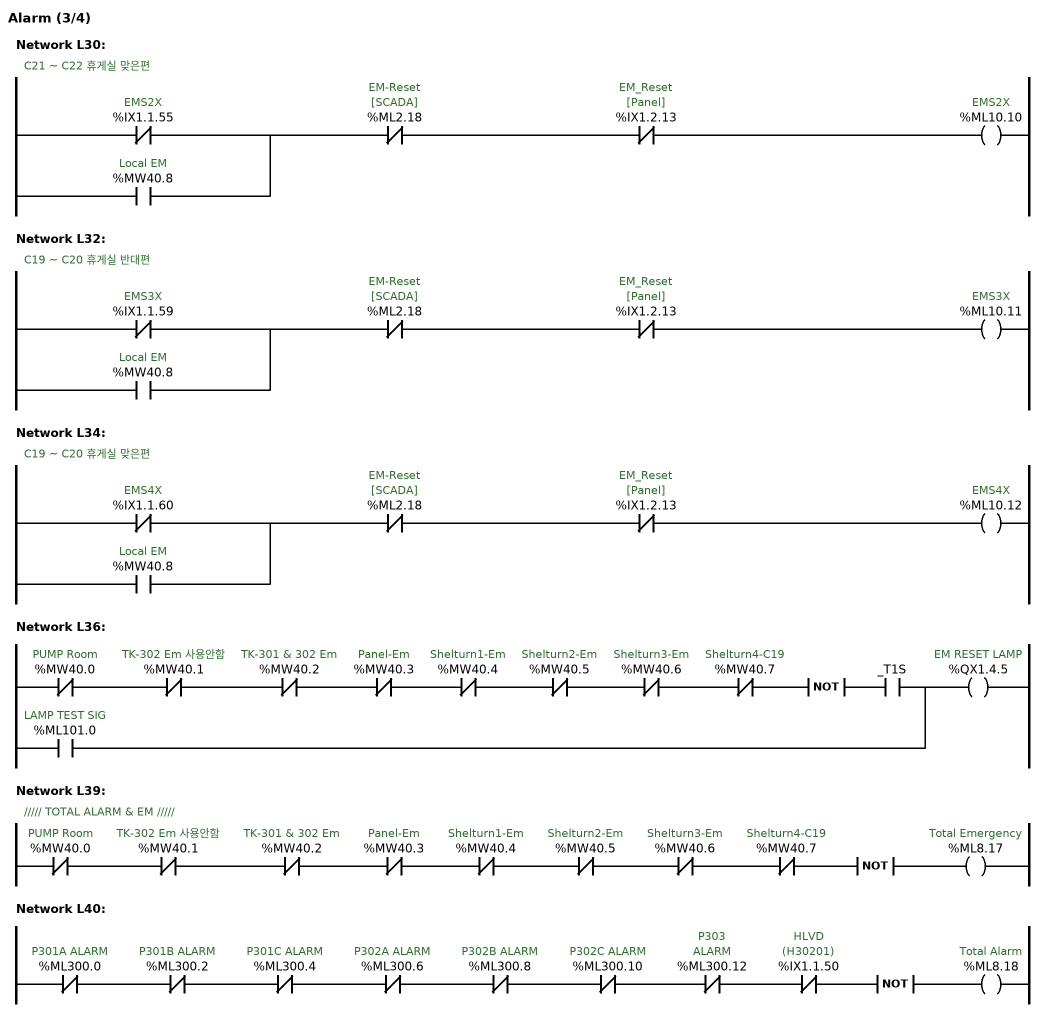
(* Rung L30 *)
%ML10.10 := (NOT %IX1.1.55 OR %MW40.8) AND NOT %ML2.18 AND NOT %IX1.2.13;
(* C21 ~ C22 휴게실 맞은편 *)
(* Rung L32 *)
%ML10.11 := (NOT %IX1.1.59 OR %MW40.8) AND NOT %ML2.18 AND NOT %IX1.2.13;
(* C19 ~ C20 휴게실 반대편 *)
(* Rung L34 *)
%ML10.12 := (NOT %IX1.1.60 OR %MW40.8) AND NOT %ML2.18 AND NOT %IX1.2.13;
(* C19 ~ C20 휴게실 맞은편 *)
(* Rung L36 *)
%QX1.4.5 := (NOT (NOT %MW40.0 AND NOT %MW40.1 AND NOT %MW40.2 AND NOT %MW40.3 AND NOT %MW40.4 AND NOT %MW40.5 AND NOT %MW40.6 AND NOT %MW40.7) AND _T1S) OR %ML101.0;
(* ///// TOTAL ALARM & EM ///// *)
(* Rung L39 *)
%ML8.17 := NOT (NOT %MW40.0 AND NOT %MW40.1 AND NOT %MW40.2 AND NOT %MW40.3 AND NOT %MW40.4 AND NOT %MW40.5 AND NOT %MW40.6 AND NOT %MW40.7);
(* Rung L40 *)
%ML8.18 := NOT (NOT %ML300.0 AND NOT %ML300.2 AND NOT %ML300.4 AND NOT %ML300.6 AND NOT %ML300.8 AND NOT %ML300.10 AND NOT %ML300.12 AND NOT %IX1.1.50);

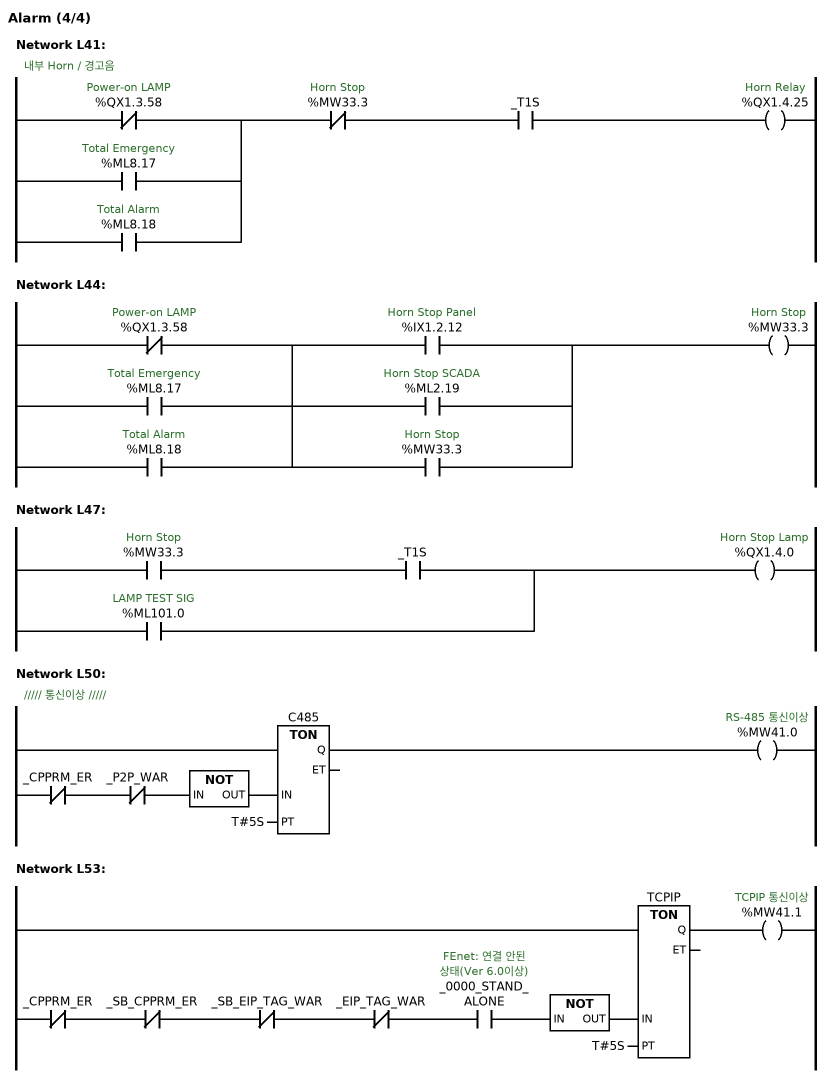
(* Rung L41 *)
%QX1.4.25 := (NOT %QX1.3.58 OR %ML8.17 OR %ML8.18) AND NOT %MW33.3 AND _T1S;
(* 내부 Horn / 경고음 *)
(* Rung L44 *)
%MW33.3 := (NOT %QX1.3.58 OR %ML8.17 OR %ML8.18) AND (%IX1.2.12 OR %ML2.19 OR %MW33.3);
(* Rung L47 *)
%QX1.4.0 := (%MW33.3 AND _T1S) OR %ML101.0;
(* ///// 통신이상 ///// *)
(* Rung L50 *)
C485(IN := NOT (NOT _CPPRM_ER AND NOT _P2P_WAR), PT := T#5S);
%MW41.0 := C485.Q;
(* Rung L53 *)
TCPIP(IN := NOT (NOT _CPPRM_ER AND NOT _SB_CPPRM_ER AND NOT _SB_EIP_TAG_WAR AND NOT _EIP_TAG_WAR AND _0000_STAND_ALONE), PT := T#5S);
%MW41.1 := TCPIP.Q;
END_PROGRAM